FUNCTION Vector_DotProduct : BOOL
VAR_INPUT
	A : REFERENCE TO Matrix;
	B : REFERENCE TO Matrix;
END_VAR
VAR_OUTPUT
	Res : LREAL;
END_VAR
VAR
	Sum : LREAL;
	I : UINT;
END_VAR

IF NOT(A.IsVector) OR NOT(B.IsVector) OR A.Length <> B.Length OR A.IsEmpty THEN
	Vector_DotProduct := FALSE;
	Res := 0;
	RETURN;
END_IF

Vector_DotProduct := TRUE;

Sum := 0;
FOR I := 0 TO A.Length-1 DO
	Sum := Sum + A.GetI(I)*B.GetI(I);
END_FOR
Res := SUM;

END_FUNCTION

(* stored: Version 1.1.0.1, ProductVersion 3.1.4024.9
   POU Vector_DotProduct: Id {ebd5ad2a-d448-0df4-1d3d-226835190fab}, SpecialFunc None *)
